FUNCTION_BLOCK FB_ClampMove
VAR_INPUT
	Ex	:BOOL;
	UnitMode	:DINT;
	paraAutoMove		:INT;
	_iHeavyGauge: INT;
END_VAR
VAR_OUTPUT
	Done	:BOOL;
END_VAR
VAR
	inMid,inFrnt,inRear,inMid2: INPUT;
	
	tonDone: Ton;
	aa: BOOL;
	iStep: INT;
	ton11: ton;
END_VAR

(*-----------------------------------------------------------------------------------*)
(*------------------------- Clamp Gauge Front/Rear/Middle ---------------------------*)
(*-----------------------------------------------------------------------------------*)


inMid(PT_OFF:=T#3S );
inFrnt(PT_OFF:=T#3S );
inRear(PT_OFF:=T#3S );
inMid2(PT_OFF:=T#3S );
CASE iStep OF
	0:
		IF stFolder.Status.Clamp_GtLowPoint AND Ex THEN
			iStep:=1;
		END_IF
	1:
	inMid.INPUT		:=Hmi_bArray[1] AND NOT In_sigGaugingMid;		//Light 			
	inFrnt.INPUT	:=NOT Hmi_bArray[1] AND _iHeavyGauge=+1 AND (NOT In_sigGaugingFrnt);//Heavy
	inRear.INPUT	:=NOT Hmi_bArray[1] AND _iHeavyGauGE=-1 AND (NOT In_sigGaugingRear);//Heavy
	inMid2.INPUT	:=NOT Hmi_bArray[1] AND _iHeavyGauGE=0  AND (NOT In_sigGaugingMid);	//Heavy Sqlusa
	IF (Hmi_bArray[1] AND In_sigGaugingMid) OR 
		(NOT Hmi_bArray[1] AND _iHeavyGauge=+1 AND In_sigGaugingFrnt) OR
		(NOT Hmi_bArray[1] AND _iHeavyGauge=-1 AND In_sigGaugingRear) OR
		(NOT Hmi_bArray[1] AND _iHeavyGauge= 0 AND In_sigGaugingMid) THEN
		iStep:=2;
	END_IF
	2:
	iStep:=3;
	3:
	iStep:=4;
	4:
	iStep:=5;
	5:
	IF NOT inFrnt.Q AND NOT inRear.Q AND NOT inMid.Q AND NOT inMid2.Q  THEN
		iStep:=10;
	END_IF
	10:
	Out_GaugingF_Ext:=Out_GaugingF_Rtn:=Out_GaugingR_Ext:=Out_GaugingR_Rtn:=FALSE;
	ton11(IN:=TRUE , PT:=T#300MS , Q=> , ET=> );
	IF ton11.Q THEN
		iStep:=11;
	END_IF
	11:
	ton11(IN:=FALSE );
	
	Done	:=TRUE;
	iStep:=0;
	Ex	:=FALSE;
	
END_CASE


	
//上钳口工作位：若Front信号未到，一直输出Front阀。直到Front信号到，延时1秒后，关闭阀。

IF inMid.Q OR inMid2.Q THEN
	Out_GaugingF_Ext:=TRUE;		Out_GaugingF_Rtn:=FALSE;	Out_GaugingR_Ext:=FALSE;	Out_GaugingR_Rtn:=TRUE;		//Middle 0mm
ELSIF inFrnt.Q THEN
	Out_GaugingF_Ext:=TRUE;		Out_GaugingF_Rtn:=FALSE;	Out_GaugingR_Ext:=TRUE;		Out_GaugingR_Rtn:=FALSE;		//Front +2MM
ELSIF inRear.Q THEN
	Out_GaugingF_Ext:=FALSE; 	Out_GaugingF_Rtn:=TRUE;		Out_GaugingR_Ext:=FALSE;	Out_GaugingR_Rtn:=TRUE;			//Rear -2MM

	
END_IF

	

tonDone(IN:=Done , PT:=T#2000MS , Q=> , ET=> );
IF tonDone.Q THEN
	Done	:=FALSE;
	
END_IF

END_FUNCTION_BLOCK

(* stored: Version 1.1.0.1, ProductVersion 3.1.4024.15
   POU FB_ClampMove: Id {d37df2b2-670f-468e-b2ba-ce0e8bd1af48}, SpecialFunc None *)
